{attribute addProperty BoxType "EL3483-0000-0016"}
{attribute addProperty Id "OvervoltageAT %I*BOOL812Inaccurate_VoltageAT %I*BOOL814Voltage_Guard_WarningAT %I*BOOL816Voltage_Guard_ErrorAT %I*BOOL817TxPDO_ToggleAT %I*BOOL8116"}
{attribute addProperty CRC "734503427"}
{attribute addProperty SizeInBites "40"}
{attribute addProperty SizeInBytes "5"}
TYPE L1_Status_2BC7A203 :
STRUCT
	{attribute addProperty Name "Overvoltage"}
	Overvoltage AT %I* : BOOL;
	{attribute addProperty Name "Inaccurate_Voltage"}
	Inaccurate_Voltage AT %I* : BOOL;
	{attribute addProperty Name "Voltage_Guard_Warning"}
	Voltage_Guard_Warning AT %I* : BOOL;
	{attribute addProperty Name "Voltage_Guard_Error"}
	Voltage_Guard_Error AT %I* : BOOL;
	{attribute addProperty Name "TxPDO_Toggle"}
	TxPDO_Toggle AT %I* : BOOL;
END_STRUCT
END_TYPE

(* stored: Version 1.2.0.0, ProductVersion 3.1.4024.9
   DUT L1_Status_2BC7A203: Id {3f807f4e-d5c7-47a4-8adf-ba99271b8985} *)
